TEXTLIST txtLstCylinderEnableMode
  0 = 'Off'
  1 = 'To Home'
  2 = 'To Out'
  3 = 'No Change Allowed'
   = ''
END_TEXTLIST

(* stored: Version 1.1.0.1, ProductVersion 3.1.4019.2
   TextList txtLstCylinderEnableMode: Id {0e302a58-7db9-4713-85a5-fe5f71396427} *)
